FUNCTION_BLOCK CROSSCOMM_PEER_21793A890546FF994 (* Service Interface Function Block Type *)
  (* Standard: 61499-2 *)
  (* Version 0.0, 9/22/2017, bababen, nxtControl GmbH, template *)
  PACKAGE Main;
  (* Compiler Cpp nxtControl builtin 1.0 *)
  {SET_ATTRIBUTE(Runtime.FBType.ImplementingType, Runtime.System#DYNGEN_CROSSCOMM_PEER)}
  {SET_ATTRIBUTE(Configuration.GenericFBType.InterfaceParams, Runtime.System#<InterfaceList> <EventOutputs> <Event Name="INITO"> <With Var="ExtendLift" /> <With Var="RetractLift" /> </Event> <Event Name="CNF"> <With Var="ExtendLift" /> <With Var="RetractLift" /> </Event> </EventOutputs> <OutputVars> <VarDeclaration Name="ExtendLift" Type="BOOL" /> <VarDeclaration Name="RetractLift" Type="BOOL" /> </OutputVars> </InterfaceList>)}
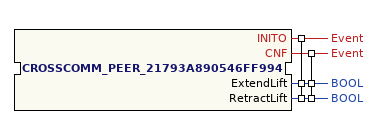
  EVENT_OUTPUT
    INITO WITH ExtendLift, RetractLift;
    CNF WITH ExtendLift, RetractLift;
  END_EVENT
  VAR_OUTPUT
    ExtendLift : BOOL;
    RetractLift : BOOL;
  END_VAR
  EC_STATES
    START;
  END_STATES
END_FUNCTION_BLOCK
